// ---- VISUs/Internal/PH_Header.TcVIS
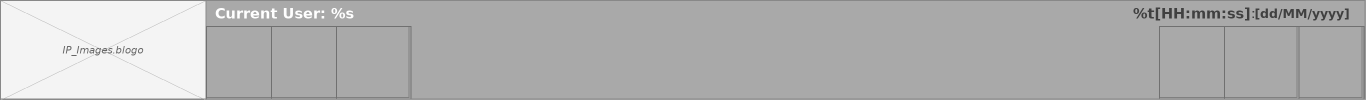
VISUALIZATION PH_Header  // 1366x100
VAR_IN_OUT
	iFrameNumber							: INT;
	bMenu 									: BOOL;
	wButton									: WORD;
END_VAR
    Button (211,34 65x65), image: IP_Buttons.menu dark
        OnMouseEnter: execute { GVL_HMI.wButton.0:=TRUE; }
        OnMouseLeave: execute { GVL_HMI.wButton.0:=FALSE; }
        OnMouseDown: execute { GVL_HMI.bMenu:=TRUE; }
    Rectangle (1233,1 120x25), "%t[dd/MM/yyyy]"
    Rectangle (212,1 250x25), "Current User: %s", text variable: VisuElemsWinControls.CurrentFullUserName
    Button (276,34 65x65), image: IP_Buttons.home dark
        OnMouseEnter: execute { GVL_HMI.wButton.1:=TRUE; }
        OnMouseLeave: execute { GVL_HMI.wButton.1:=FALSE; }
        OnMouseDown: execute { GVL_HMI.iFrameNumber:=0; GVL_HMI.bMenu:=FALSE; }
    Button (341,34 65x65), image: IP_Buttons.alarms dark
        OnMouseEnter: execute { GVL_HMI.wButton.2:=TRUE; }
        OnMouseLeave: execute { GVL_HMI.wButton.2:=False; }
        OnMouseDown: execute { GVL_HMI.iFrameNumber:=1; GVL_HMI.bMenu:=FALSE; }
    Button (1164,34 65x65), image: IP_Buttons.info dark
        OnMouseEnter: execute { GVL_HMI.wButton.3:=TRUE; }
        OnMouseLeave: execute { GVL_HMI.wButton.3:=FALSE; }
        OnMouseDown: execute { GVL_HMI.iFrameNumber:=2; GVL_HMI.bMenu:=FALSE; }
    Button (1229,34 65x65), colour toggle: GVL_HMI.wButton.4, image: IP_Buttons.user dark
        OnMouseEnter: execute { GVL_HMI.wButton.4:=TRUE; }
        OnMouseLeave: execute { GVL_HMI.wButton.4:=FALSE; }
        OnMouseDown: execute { GVL_HMI.iFrameNumber:=3; GVL_HMI.bMenu:=FALSE; }
    Button (1294,34 65x65), image: IP_Buttons.set dark
        OnMouseEnter: execute { GVL_HMI.wButton.5:=TRUE; }
        OnMouseLeave: execute { GVL_HMI.wButton.5:=FALSE; }
        OnMouseDown: execute { GVL_HMI.iFrameNumber:=4; GVL_HMI.bMenu:=FALSE; }
    Rectangle (1132,1 120x25), "%t[HH:mm:ss]"
    RoundedRectangle (625,53 280x40), text list: 'TL_Frames', text index: iFrameNumber
    Image (0,0 206x100), image: IP_Images.blogo
    Button (1229,34 65x65), invisible if: NOT GVL_HMI.wButton.4, image: IP_Buttons.user light
        OnMouseEnter: execute { GVL_HMI.wButton.4:=TRUE; }
        OnMouseLeave: execute { GVL_HMI.wButton.4:=FALSE; }
        OnMouseDown: execute { GVL_HMI.iFrameNumber:=3; GVL_HMI.bMenu:=FALSE; }
    Button (1294,34 65x65), invisible if: NOT GVL_HMI.wButton.5, image: IP_Buttons.set light
        OnMouseEnter: execute { GVL_HMI.wButton.5:=TRUE; }
        OnMouseLeave: execute { GVL_HMI.wButton.5:=FALSE; }
        OnMouseDown: execute { GVL_HMI.iFrameNumber:=4; GVL_HMI.bMenu:=FALSE; }
    Button (1289,26 75x73), invisible if: iFrameNumber<>4 OR GVL_HMI.bMenu, image: IP_Buttons.set dark
        OnMouseEnter: execute { GVL_Hmi.wButton.5:=TRUE; }
        OnMouseLeave: execute { GVL_Hmi.wButton.5:=FALSE; }
    Button (1289,26 75x73), invisible if: iFrameNumber<>4 OR GVL_HMI.bMenu OR NOT GVL_HMI.wButton.5, image: IP_Buttons.set light
        OnMouseEnter: execute { GVL_Hmi.wButton.5:=TRUE; }
        OnMouseLeave: execute { GVL_Hmi.wButton.5:=FALSE; }
    Button (1164,34 65x65), invisible if: NOT GVL_HMI.wButton.3, image: IP_Buttons.info light
        OnMouseEnter: execute { GVL_HMI.wButton.3:=TRUE; }
        OnMouseLeave: execute { GVL_HMI.wButton.3:=FALSE; }
        OnMouseDown: execute { GVL_HMI.iFrameNumber:=2; GVL_HMI.bMenu:=FALSE; }
    Button (1159,26 75x73), invisible if: iFrameNumber<>2 OR GVL_HMI.bMenu, image: IP_Buttons.info dark
        OnMouseEnter: execute { GVL_Hmi.wButton.3:=TRUE; }
        OnMouseLeave: execute { GVL_Hmi.wButton.3:=FALSE; }
    Button (1159,26 75x73), invisible if: iFrameNumber<>2 OR GVL_HMI.bMenu OR NOT GVL_HMI.wButton.3, image: IP_Buttons.info light
        OnMouseEnter: execute { GVL_Hmi.wButton.3:=TRUE; }
        OnMouseLeave: execute { GVL_Hmi.wButton.3:=FALSE; }
    Button (341,34 65x65), invisible if: NOT GVL_HMI.wButton.2, image: IP_Buttons.alarms light
        OnMouseEnter: execute { GVL_HMI.wButton.2:=TRUE; }
        OnMouseLeave: execute { GVL_HMI.wButton.2:=False; }
        OnMouseDown: execute { GVL_HMI.iFrameNumber:=1; GVL_HMI.bMenu:=FALSE; }
    Button (276,34 65x65), invisible if: NOT GVL_HMI.wButton.1, image: IP_Buttons.home light
        OnMouseEnter: execute { GVL_HMI.wButton.1:=TRUE; }
        OnMouseLeave: execute { GVL_HMI.wButton.1:=FALSE; }
        OnMouseDown: execute { GVL_HMI.iFrameNumber:=0; GVL_HMI.bMenu:=FALSE; }
    Button (1224,26 75x73), invisible if: iFrameNumber<>3 OR GVL_HMI.bMenu, image: IP_Buttons.user dark
        OnMouseEnter: execute { GVL_Hmi.wButton.4:=TRUE; }
        OnMouseLeave: execute { GVL_Hmi.wButton.4:=FALSE; }
    Button (1224,26 75x73), invisible if: iFrameNumber<>3 OR GVL_HMI.bMenu OR NOT GVL_HMI.wButton.4, image: IP_Buttons.user light
        OnMouseEnter: execute { GVL_Hmi.wButton.4:=TRUE; }
        OnMouseLeave: execute { GVL_Hmi.wButton.4:=FALSE; }
    Button (211,34 65x65), invisible if: NOT GVL_HMI.wButton.0, image: IP_Buttons.menu light
        OnMouseEnter: execute { GVL_HMI.wButton.0:=TRUE; }
        OnMouseLeave: execute { GVL_HMI.wButton.0:=FALSE; }
        OnMouseDown: execute { GVL_HMI.bMenu:=TRUE; }
    Button (206,26 75x73), invisible if: NOT GVL_HMI.bMenu, image: IP_Buttons.menu dark
        OnMouseEnter: execute { GVL_Hmi.wButton.0:=TRUE; }
        OnMouseLeave: execute { GVL_Hmi.wButton.0:=FALSE; }
    Button (206,26 75x73), invisible if: NOT GVL_HMI.bMenu OR NOT GVL_HMI.wButton.0, image: IP_Buttons.menu light
        OnMouseEnter: execute { GVL_Hmi.wButton.0:=TRUE; }
        OnMouseLeave: execute { GVL_Hmi.wButton.0:=FALSE; }
    Button (271,26 75x73), invisible if: iFrameNumber<>0 OR GVL_HMI.bMenu, image: IP_Buttons.home dark
        OnMouseEnter: execute { GVL_Hmi.wButton.1:=TRUE; }
        OnMouseLeave: execute { GVL_Hmi.wButton.1:=FALSE; }
    Button (271,26 75x73), invisible if: iFrameNumber<>0 OR GVL_HMI.bMenu OR NOT GVL_HMI.wButton.1, image: IP_Buttons.home light
        OnMouseEnter: execute { GVL_Hmi.wButton.1:=TRUE; }
        OnMouseLeave: execute { GVL_Hmi.wButton.1:=FALSE; }
    Button (336,26 75x73), invisible if: iFrameNumber<>1 OR GVL_HMI.bMenu, image: IP_Buttons.alarms dark
        OnMouseEnter: execute { GVL_Hmi.wButton.2:=TRUE; }
        OnMouseLeave: execute { GVL_Hmi.wButton.2:=FALSE; }
    Button (336,26 75x73), invisible if: iFrameNumber<>1 OR GVL_HMI.bMenu OR NOT GVL_HMI.wButton.2, image: IP_Buttons.alarms light
        OnMouseEnter: execute { GVL_Hmi.wButton.2:=TRUE; }
        OnMouseLeave: execute { GVL_Hmi.wButton.2:=FALSE; }
END_VISUALIZATION

// ---- VISUs/Internal/PH_Menu.TcVIS
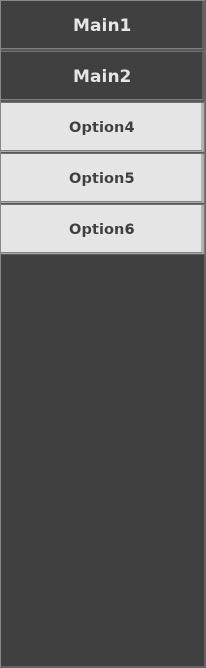
VISUALIZATION PH_Menu  // 206x668
VAR_IN_OUT
	bMain1									: BOOL;
	bMain2									: BOOL;
	iFrameNumber							: INT;
	udiFOntColor1 							: UDINT;
	udiFontColor2							: UDINT;
END_VAR
    Group (0,0 206x254), invisible if: NOT GVL_HMI.bMenu
        Group (0,51 206x152), invisible if: NOT bMain1
            Button (0,0 204x50), "File Dialog"
                OnMouseDown: execute { GVL_HMI.iFrameNumber:=5; GVL_HMI.bMenu:=FALSE; }
            Button (0,102 204x50), "Trends"
                OnMouseDown: execute { GVL_HMI.iFrameNumber:=7; GVL_HMI.bMenu:=FALSE; }
            Button (0,51 204x50), "Table"
                OnMouseDown: execute { GVL_HMI.iFrameNumber:=6; GVL_HMI.bMenu:=FALSE; }
        Group (0,102 206x152), invisible if: NOT bMain2
            Button (0,102 204x50), "Option6"
                OnMouseDown: execute { GVL_HMI.iFrameNumber:=10; GVL_HMI.bMenu:=FALSE; }
            Button (0,51 204x50), "Option5"
                OnMouseDown: execute { GVL_HMI.iFrameNumber:=9; GVL_HMI.bMenu:=FALSE; }
            Button (0,0 204x50), "Option4"
                OnMouseDown: execute { GVL_HMI.iFrameNumber:=8; GVL_HMI.bMenu:=FALSE; }
        Button (0,51 205x50), "Main2", colour toggle: bMain2
            p2738717112: BOOL_TO_INT(bMain1)*153
            p55702900: udiFontColor2
            OnMouseDown: execute { GVL_Hmi.bMain1:=FALSE; GVL_HMI.bMain2:=TRUE; }
        Button (0,0 205x50), "Main1", colour toggle: bMain1
            p55702900: udiFOntColor1
            OnMouseDown: execute { GVL_HMI.bMain2:=FALSE; GVL_HMI.bMain1:=TRUE; }
END_VISUALIZATION

// ---- VISUs/Internal/PH_SystemInfo.TcVIS
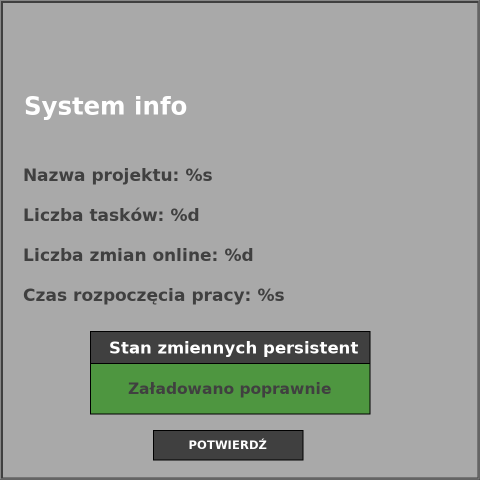
VISUALIZATION PH_SystemInfo  // 480x480
VAR
	bConfirmButtonState						: BOOL:=FALSE;
END_VAR
    Rectangle (0,0 480x480)
    Rectangle (90,331 280x83)
    Label (21,91 175x30), "System info"
    Rectangle (20,160 339x30), "Nazwa projektu: %s", text variable: _AppInfo.ProjectName
    Rectangle (20,200 339x30), "Liczba tasków: %d", text variable: _AppInfo.TaskCnt
    Rectangle (20,240 339x30), "Liczba zmian online: %d", text variable: _AppInfo.OnlineChangeCnt
    Rectangle (20,280 437x30), "Czas rozpoczęcia pracy: %s", text variable: P_SystemInfo.sStartTime
    RoundedRectangle (153,430 150x30), "POTWIERDŹ", colour toggle: bConfirmButtonState
        OnMouseUp: execute { bConfirmButtonState:=FALSE; }
        OnMouseUp: execute { P_SystemInfo.bConfirm:=FALSE; }
        OnMouseLeave: execute { bConfirmButtonState:=FALSE; }
        OnMouseLeave: execute { P_SystemInfo.bConfirm:=FALSE; }
        OnMouseDown: execute { bConfirmButtonState:=TRUE; }
        OnMouseDown: execute { P_SystemInfo.bConfirm:=TRUE; }
    Rectangle (95,333 258x30), "Stan zmiennych persistent"
    Rectangle (90,363 280x51), "Błąd", invisible if: NOT P_SystemInfo.bError
    Rectangle (90,363 280x51), "Załadowano plik zapasowy", invisible if: NOT P_SystemInfo.bWarning
    Rectangle (90,363 280x51), "Załadowano poprawnie", invisible if: NOT P_SystemInfo.bOK
END_VISUALIZATION

// ---- VISUs/Internal/PH_TaskInfo.TcVIS
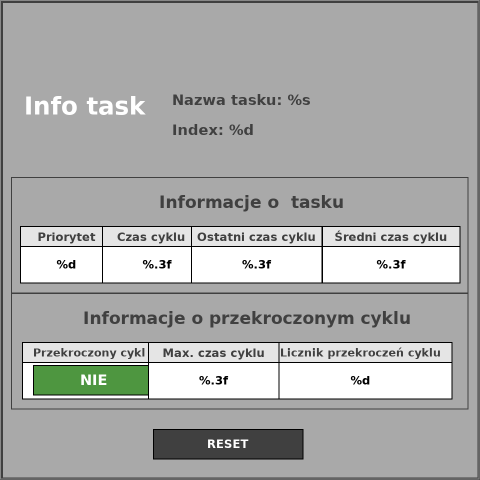
VISUALIZATION PH_TaskInfo  // 480x480
VAR_IN_OUT
	fbTaskInfo								: FB_TaskInfo;
	bReset									: BOOL;
END_VAR
VAR

END_VAR
    Rectangle (0,0 480x480)
    Label (21,91 150x30), "Info task"
    RoundedRectangle (11,177 457x116)
    Label (156,187 185x30), "Informacje o tasku"
    Rectangle (169,85 307x30), "Nazwa tasku: %s", text variable: fbTaskInfo.sTaskName
    Rectangle (169,115 150x30), "Index: %d", text variable: fbTaskInfo.byIndex
    RoundedRectangle (11,293 457x116)
    Label (80,303 320x30), "Informacje o przekroczonym cyklu"
    Group (20,226 82x57)
        RoundedRectangle (0,0 93x22), "Priorytet"
        Rectangle (0,20 93x37), "%d", text variable: fbTaskInfo.uiPriority
    RoundedRectangle (20,226 93x22), "Priorytet"
    Rectangle (20,246 93x37), "%d", text variable: fbTaskInfo.uiPriority
    Group (269,342 183x57)
        RoundedRectangle (0,0 183x22), "Licznik przekroczeń cyklu"
        Rectangle (0,20 183x37), "%d", text variable: fbTaskInfo.udiCountExceedCycle
    RoundedRectangle (269,342 183x22), "Licznik przekroczeń cyklu"
    Rectangle (269,362 183x37), "%d", text variable: fbTaskInfo.udiCountExceedCycle
    Group (22,342 126x57)
        RoundedRectangle (0,0 144x22), "Przekroczony cykl"
        Rectangle (0,20 144x37)
        RoundedRectangle (11,23 122x30), "TAK"
        RoundedRectangle (11,23 122x30), "NIE", invisible if: fbTaskInfo.bCycleTimeExceeded
    RoundedRectangle (22,342 144x22), "Przekroczony cykl"
    Rectangle (22,362 144x37)
    RoundedRectangle (33,365 122x30), "TAK"
    RoundedRectangle (33,365 122x30), "NIE", invisible if: fbTaskInfo.bCycleTimeExceeded
    Group (102,226 89x57)
        RoundedRectangle (0,0 110x22), "Czas cyklu"
        Rectangle (0,20 110x37), "%.3f", text variable: fbTaskInfo.rCycleTime
    RoundedRectangle (102,226 110x22), "Czas cyklu"
    Rectangle (102,246 110x37), "%.3f", text variable: fbTaskInfo.rCycleTime
    Group (191,226 131x57)
        RoundedRectangle (0,0 131x22), "Ostatni czas cyklu"
        Rectangle (0,20 131x37), "%.3f", text variable: fbTaskInfo.rLastExecTime
    RoundedRectangle (191,226 131x22), "Ostatni czas cyklu"
    Rectangle (191,246 131x37), "%.3f", text variable: fbTaskInfo.rLastExecTime
    Group (322,226 128x57)
        RoundedRectangle (0,0 138x22), "Średni czas cyklu"
        Rectangle (0,20 138x37), "%.3f", text variable: fbTaskInfo.rAverageCycleTime
    RoundedRectangle (322,226 138x22), "Średni czas cyklu"
    Rectangle (322,246 138x37), "%.3f", text variable: fbTaskInfo.rAverageCycleTime
    Group (148,342 121x57)
        RoundedRectangle (0,0 131x22), "Max. czas cyklu"
        Rectangle (0,20 131x37), "%.3f", text variable: fbTaskInfo.rMaxExecTime
    RoundedRectangle (148,342 131x22), "Max. czas cyklu"
    Rectangle (148,362 131x37), "%.3f", text variable: fbTaskInfo.rMaxExecTime
    RoundedRectangle (153,429 150x30), "RESET", colour toggle: bReset
        tap bReset
END_VISUALIZATION

// ---- VISUs/Menus/V_FileDialog.TcVIS
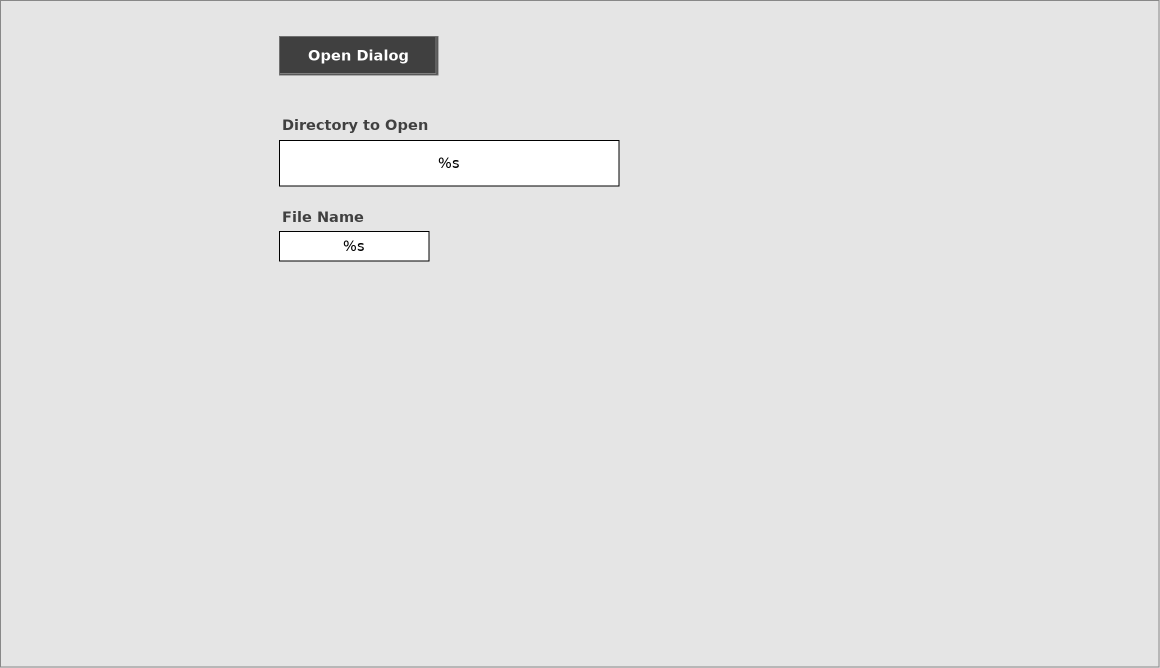
VISUALIZATION V_FileDialog  // 1160x668
    Button (279,36 159x39), "Open Dialog"
        tap P_FileDialog.bOpen
        OnMouseDown: OpenDialog Dialog=VisuDialogs.FileOpenSave, Parameters={fileListProvider: P_FileDialog.fbFileList}, OpenModal=True, OpenCentered=True
    Rectangle (279,231 150x30), "%s", text variable: P_FileDialog.sSelectedFileName
    Textfield (279,140 340x46), "%s", text variable: P_FileDialog.sDir
        OnMouseClick: write the text variable via Edit
    Label (279,107 264x36), "Directory to Open"
    Label (279,199 264x36), "File Name"
END_VISUALIZATION

// ---- VISUs/Menus/V_Option6.TcVIS
VISUALIZATION V_Option6  // 1160x668
END_VISUALIZATION

// ---- VISUs/Menus/V_Table.TcVIS
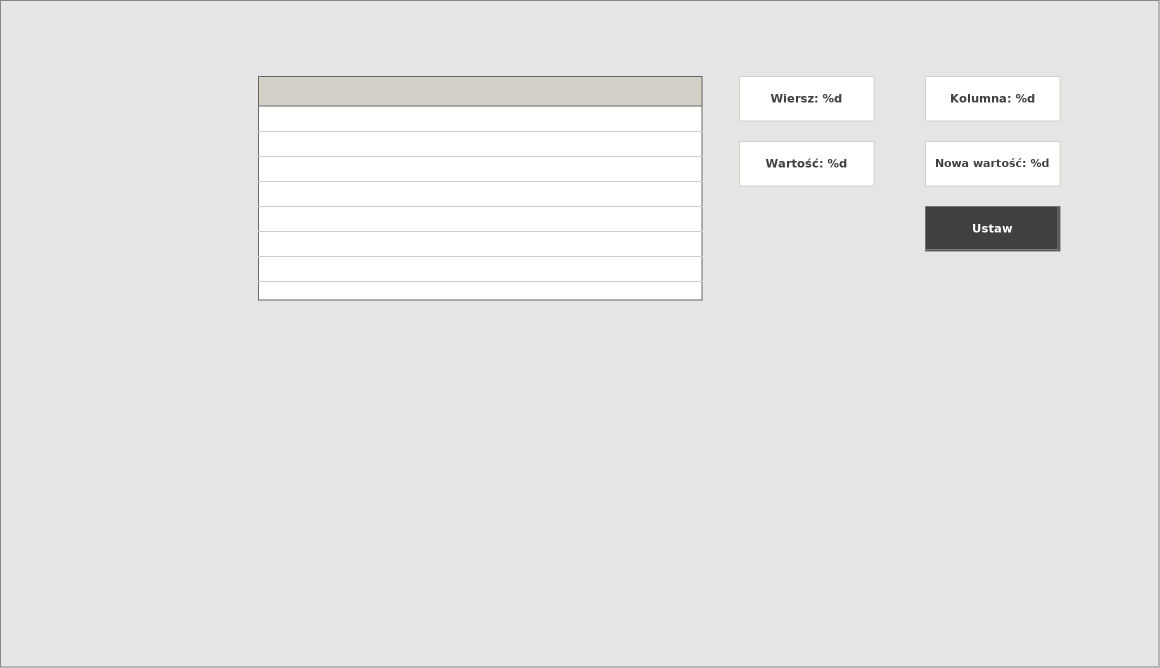
VISUALIZATION V_Table  // 1160x668
VAR_IN_OUT
	arrTable 								: ARRAY[1..10,1..10] OF INT;
	iColumn 								: INT;
	iLine 									: INT;
	iValue									: INT;
	iSetValue								: INT;
	bSet									: BOOL;
END_VAR
    Table (258,76 444x224), data array: arrTable
        p3854506369: arrTable[1,INDEX]
        p1892666644: arrTable[2,INDEX]
        p338671338: arrTable[3,INDEX]
        p2170511999: arrTable[4,INDEX]
        p3723444502: arrTable[5,INDEX]
        p1218418051: arrTable[6,INDEX]
        p746581629: arrTable[7,INDEX]
        p3104783080: arrTable[8,INDEX]
        p2501879983: arrTable[9,INDEX]
        p7306298: arrTable[10,INDEX]
        p1420305297: P_Table.iColumn
        p1137915858: P_Table.iLine
    Textfield (739,76 135x45), "Wiersz: %d", text variable: iLine
    Textfield (925,76 135x45), "Kolumna: %d", text variable: iColumn
    Textfield (739,141 135x45), "Wartość: %d", text variable: iValue
    Textfield (925,141 135x45), "Nowa wartość: %d", text variable: iSetValue
        OnMouseDown: write the text variable via Edit
    Button (925,206 135x45), "Ustaw"
        tap bSet
END_VISUALIZATION

// ---- VISUs/Menus/V_Trend.TcVIS
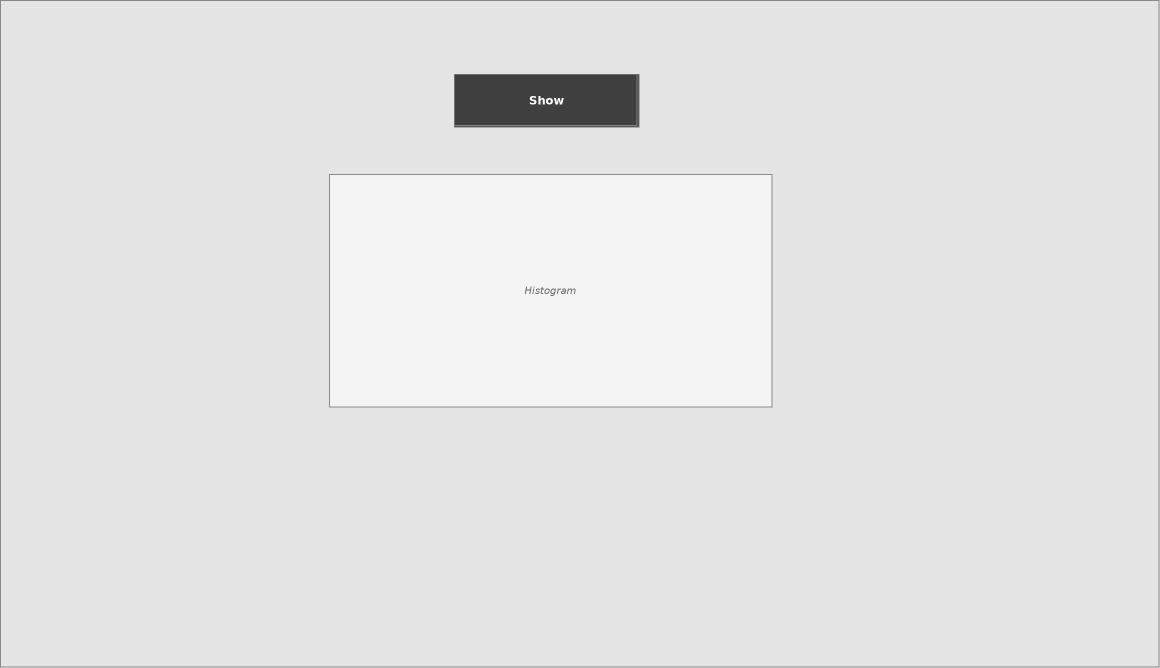
VISUALIZATION V_Trend  // 1160x668
VAR_IN_OUT
	arrHistogram 							: ARRAY [1..20] OF INT;
	bShow 									: BOOL;
END_VAR
    Histogram (329,174 443x233), scale format: %.1f, scale 0..40
        p1518820177: arrHistogram
        p102497268: arrHistogram
        p788070771: ARRAY [1..20] OF INT
    Button (454,74 185x53), "Show", colour toggle: bShow
        toggle bShow
END_VISUALIZATION

// ---- VISUs/Menus/V_Option4.TcVIS
VISUALIZATION V_Option4  // 1160x668
END_VISUALIZATION

// ---- VISUs/Menus/V_Option5.TcVIS
VISUALIZATION V_Option5  // 1160x668
END_VISUALIZATION

// ---- VISUs/TL_Frames.TcTLO
TEXTLIST TL_Frames
  0 = 'Home' | EN\: 'Home' | PL: 'Główna'
  1 = 'Alarms' | EN\: 'Alarms' | PL: 'Alarmy'
  2 = 'Info' | EN\: 'Info' | PL: 'Info'
  3 = 'Users' | EN\: 'Users' | PL: 'Użytkownicy'
  4 = 'Settings' | EN\: 'Settings' | PL: 'Ustawienia'
  5 = 'File Dialog' | EN\: 'File Dialog' | PL: 'Dialog plików'
  6 = 'Table' | EN\: 'Table' | PL: 'Tabela'
  7 = 'Trends' | EN\: 'Trends' | PL: 'Trendy'
  8 = 'Option4' | EN\: 'Option4' | PL: 'Opcja4'
  9 = 'Option5' | EN\: 'Option5' | PL: 'Opcja5'
  10 = 'Option6' | EN\: 'Opion6' | PL: 'Opcja6'
   = ''
END_TEXTLIST

// ---- VISUs/TL_Lang.TcTLO
TEXTLIST TL_Lang
  0 = 'English' | EN\: 'English' | EN: 'English' | PL: 'Angielski' | PL\: 'Angielski'
  1 = 'Polish' | EN\: 'Polish' | EN: 'Polish' | PL: 'Polski' | PL\: 'Polski'
   = ''
END_TEXTLIST

// ---- VISUs/Visualization.TcVIS
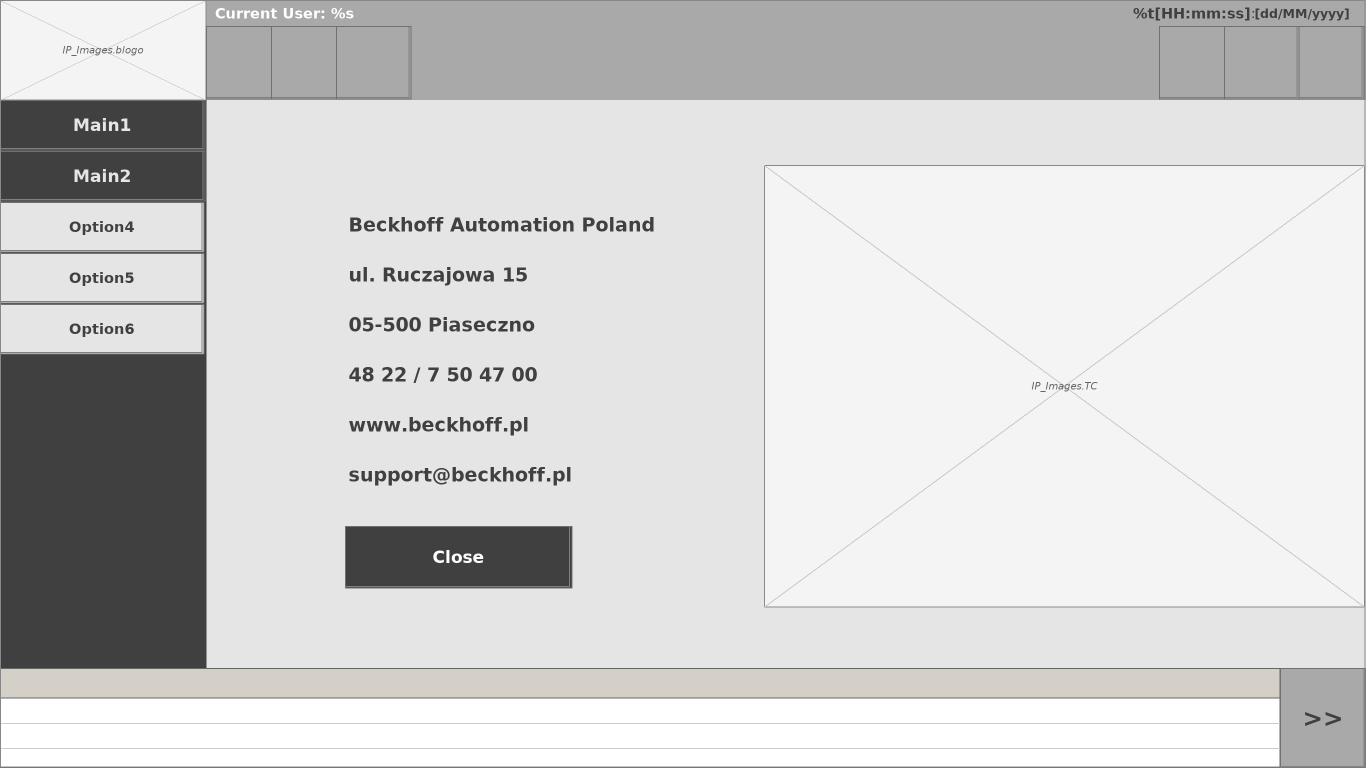
VISUALIZATION Visualization  // 1366x768
    Frame (0,0 1366x100)
        shows PH_Header(iFrameNumber := GVL_HMI.iFrameNumber, bMenu := GVL_HMI.bMenu, wButton := GVL_HMI.wButton)
    Frame (0,100 1366x668), frame switch variable: GVL_HMI.iFrameNumber
        shows V_Home(bKillProcess := P_CloseTcHmiExe.bKillProcess, sImageOsName := P_ControllerInfo.stDevIdent.strImageOsName)
        shows V_EventsHistoricalSimple()
        shows V_info()
        shows V_Users()
        shows V_Settings()
        shows V_FileDialog()
        shows V_Table(arrTable := P_Table.arrTable, iColumn := P_Table.iColumn, iLine := P_Table.iLine, iValue := P_Table.iValue, iSetValue := P_Table.iSetValue, bSet := P_Table.bSetNewValue)
        shows V_Trend(arrHistogram := P_Table.arrHistogram, bShow := P_Table.bRotate)
        shows V_Option4()
        shows V_Option5()
        shows V_Option6()
    Frame (0,100 206x668), invisible if: NOT GVL_HMI.bMenu
        shows PH_Menu(bMain1 := GVL_HMI.bMain1, bMain2 := GVL_HMI.bMain2, iFrameNumber := GVL_HMI.iFrameNumber, udiFOntColor1 := GVL_HMI.udiFOntColor1, udiFontColor2 := GVL_HMI.udiFOntColor2)
    Frame (0,668 1366x100), invisible if: GVL_HMI.iFrameNumber=1
        shows PH_Bottom(bReset := GVL_HMI.bReset, arrEventVisu := GVL_EHS.arrEventVisu)
END_VISUALIZATION

// ---- VISUs/V_EventsHistoricalSimple.TcVIS
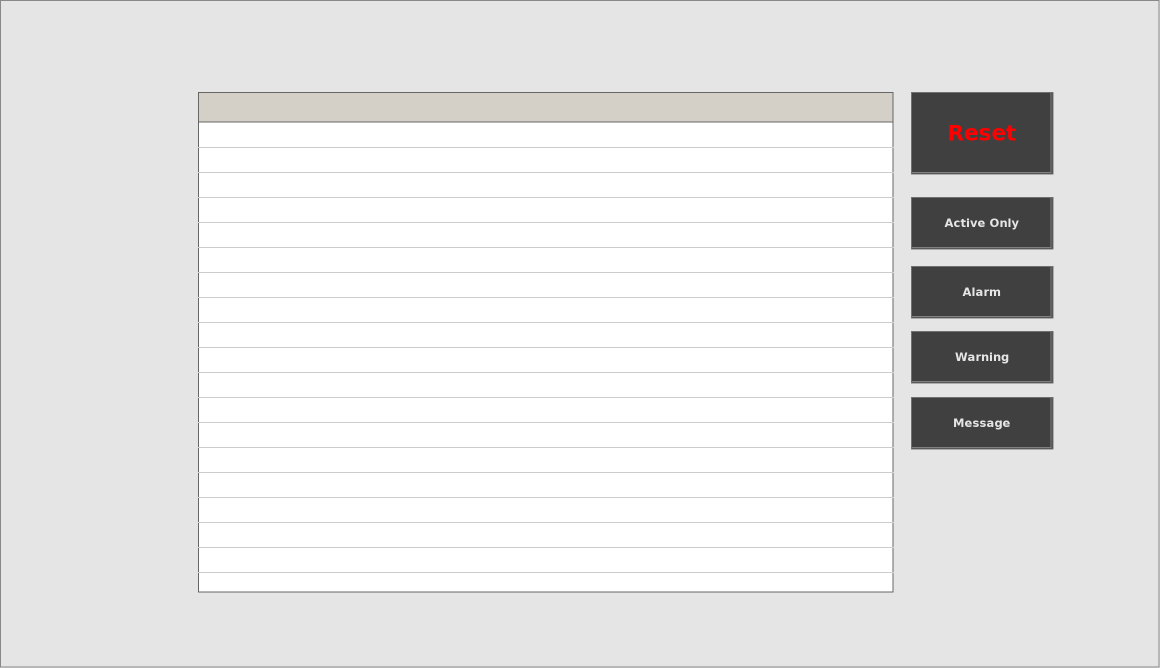
VISUALIZATION V_EventsHistoricalSimple  // 1160x668
    Table (198,92 695x500), data array: GVL_EHS.arrEventVisu
        p3854506369: GVL_EHS.arrEventVisu[INDEX].dwID
        p505689113: Date End
        p1218418051: GVL_EHS.arrEventVisu[INDEX].dtDateEnd
        p2237128397: Date Begin
        p3723444502: GVL_EHS.arrEventVisu[INDEX].dtDateBegin
        p511219082: Class
        p1892666644: GVL_EHS.arrEventVisu[INDEX].dwClass
        p1755163831: Message
        p338671338: GVL_EHS.arrEventVisu[INDEX].wsMessage
        p4092479075: Param
        p2170511999: GVL_EHS.arrEventVisu[INDEX].dwParam
        Columns.Column.[4].Template: GVL_EHS.arrEventVisu[INDEX].dwColor
        Columns.Column.[2].Template: GVL_EHS.arrEventVisu[INDEX].dwColor
        Columns.Column.[1].Template: GVL_EHS.arrEventVisu[INDEX].dwColor
        Columns.Column.[0].Template: GVL_EHS.arrEventVisu[INDEX].dwColor
        Columns.Column.[3].Template: GVL_EHS.arrEventVisu[INDEX].dwColor
        Columns.Column.[5].Template: GVL_EHS.arrEventVisu[INDEX].dwColor
    Button (911,197 142x52), "Active Only", colour toggle: P_EventsVisu.bFilterActiveOnly
        toggle P_EventsVisu.bFilterActiveOnly
    Button (911,92 142x82), "Reset"
    Button (911,266 142x52), "Alarm"
        tap GVL_HMI.bAlarm
    Button (911,331 142x52), "Warning"
        tap GVL_HMI.bWarning
    Button (911,397 142x52), "Message"
        tap GVL_HMI.bMessage
END_VISUALIZATION

// ---- VISUs/V_Home.TcVIS
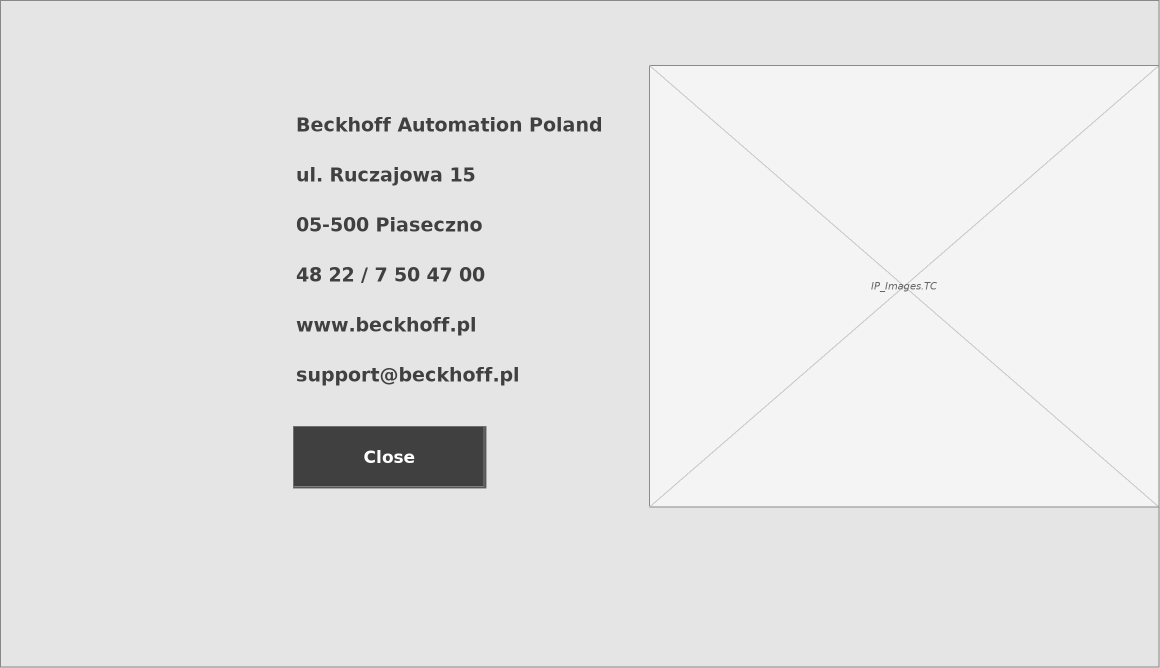
VISUALIZATION V_Home  // 1160x668
VAR_IN_OUT
	bKillProcess							: BOOL;
	sImageOsName							: STRING(20);
END_VAR
    Label (293,100 360x50), "Beckhoff Automation Poland"
    Label (293,150 360x50), "ul. Ruczajowa 15"
    Label (293,200 360x50), "05-500 Piaseczno"
    Label (293,250 360x50), "48 22 / 7 50 47 00"
    Label (293,300 360x50), "www.beckhoff.pl"
    Label (293,350 360x50), "support@beckhoff.pl"
    Image (649,65 510x442), image: IP_Images.TC
    Button (293,426 193x62), "Close", invisible if: sImageOsName='Windows CE'
        tap bKillProcess
END_VISUALIZATION

// ---- VISUs/V_info.TcVIS
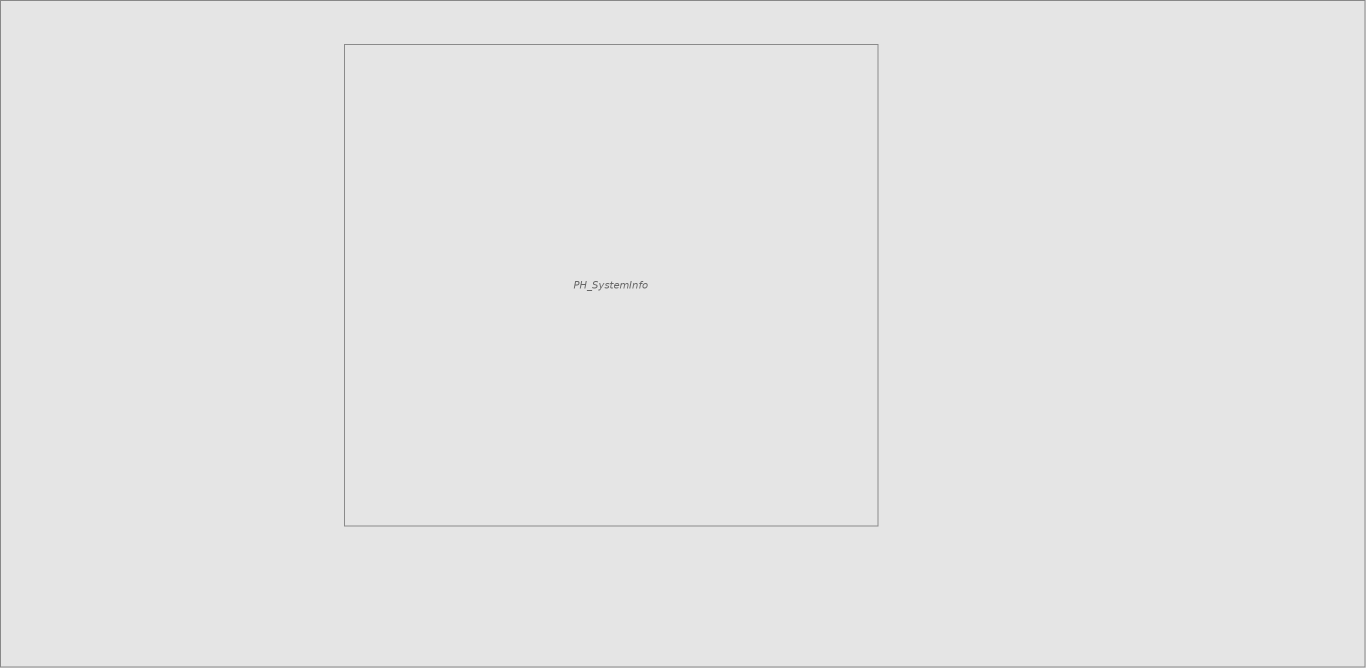
VISUALIZATION V_info  // 1366x668
    TabControl (344,44 534x482)
        shows PH_SystemInfo()
        shows PH_TaskInfo(fbTaskInfo := P_TaskInfo.fbTaskInfo, bReset := P_TaskInfo.fbTaskInfo.bResetVisu)
        shows PH_ControllerInfo(strTargetType := P_ControllerInfo.stDevIdent.strTargetType, strHardwareModel := P_ControllerInfo.stDevIdent.strHardwareModel, strHardwareSerialNo := P_ControllerInfo.stDevIdent.strHardwareSerialNo, strHardwareVersion := P_ControllerInfo.stDevIdent.strHardwareVersion, strHardwareDate := P_ControllerInfo.stDevIdent.strHardwareDate, strHardwareCPU := P_ControllerInfo.stDevIdent.strHardwareCPU, strImageDevice := P_ControllerInfo.stDevIdent.strImageDevice, strImageVersion := P_ControllerInfo.stDevIdent.strImageVersion, strImageLevel := P_ControllerInfo.stDevIdent.strImageLevel, strImageOsName := P_ControllerInfo.stDevIdent.strImageOsName, strImageOsVersion := P_ControllerInfo.stDevIdent.strImageOsVersion, strTwinCATVersion := P_ControllerInfo.stDevIdent.strTwinCATVersion, strTwinCATRevision := P_ControllerInfo.stDevIdent.strTwinCATRevision, strTwinCATBuild := P_ControllerInfo.stDevIdent.strTwinCATBuild, strTwinCATLevel := P_ControllerInfo.stDevIdent.strTwinCATLevel, strAmsNetId := P_ControllerInfo.stDevIdent.strAmsNetId, arrDevIdent := P_ControllerInfo.arrDevIdent, wDeviceInfo := GVL_HMI.wDeviceInfo, iSelectedRow := P_ControllerInfo.iSelectedRow)
        [0]: TabTitle=System Info
        [1]: TabTitle=Task Info
        [2]: TabTitle=Device Info
END_VISUALIZATION

// ---- VISUs/V_Settings.TcVIS
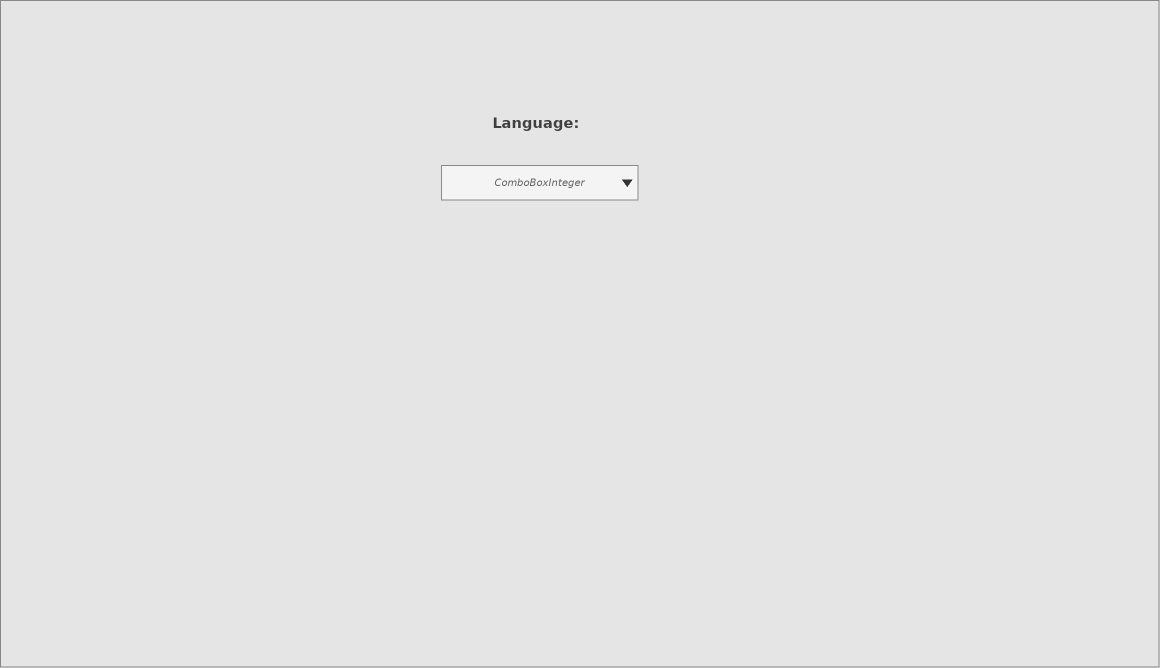
VISUALIZATION V_Settings  // 1160x668
    ComboBoxInteger (441,165 197x35), variable: GVL_HMI.iLang, text list: 'TL_Lang'
    Rectangle (443,100 186x46), "Language:"
END_VISUALIZATION

// ---- VISUs/V_Users.TcVIS
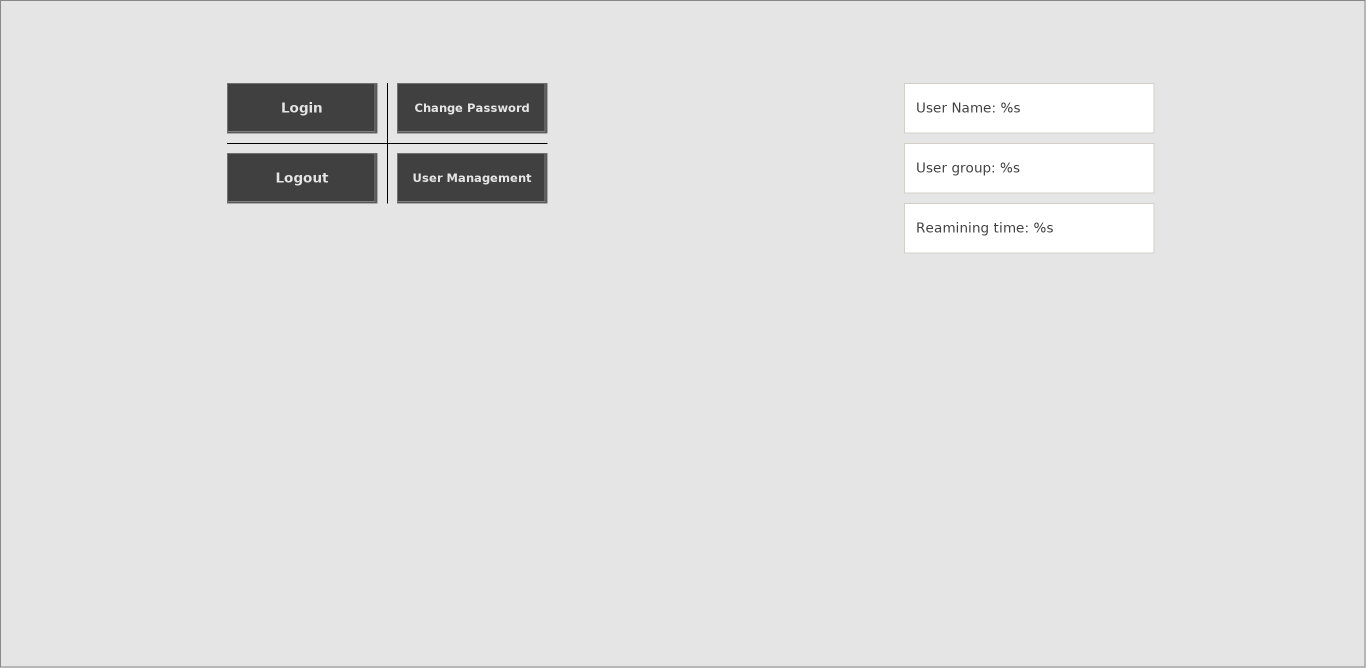
VISUALIZATION V_Users  // 1366x668
    Button (227,83 150x50), "Login"
        OnMouseDown: VisuUserMgmt Type=Login
    Button (227,153 150x50), "Logout"
        OnMouseDown: VisuUserMgmt Type=Logout
    Button (397,83 150x50), "Change Password"
        OnMouseDown: VisuUserMgmt Type=ChangeUserPassword
    Button (397,153 150x50), "User Management"
        OnMouseDown: VisuUserMgmt Type=OpenUserConfiguration
    Line (387,83) (387,203)
    Line (227,143) (547,143)
    Textfield (904,83 250x50), "User Name: %s", text variable: VisuElemsWinControls.CurrentUserName
    Textfield (904,143 250x50), "User group: %s", text variable: VisuElemsWinControls.CurrentUserGroupName
    Textfield (904,203 250x50), "Reamining time: %s", text variable: P_UserControl.sTime
END_VISUALIZATION
